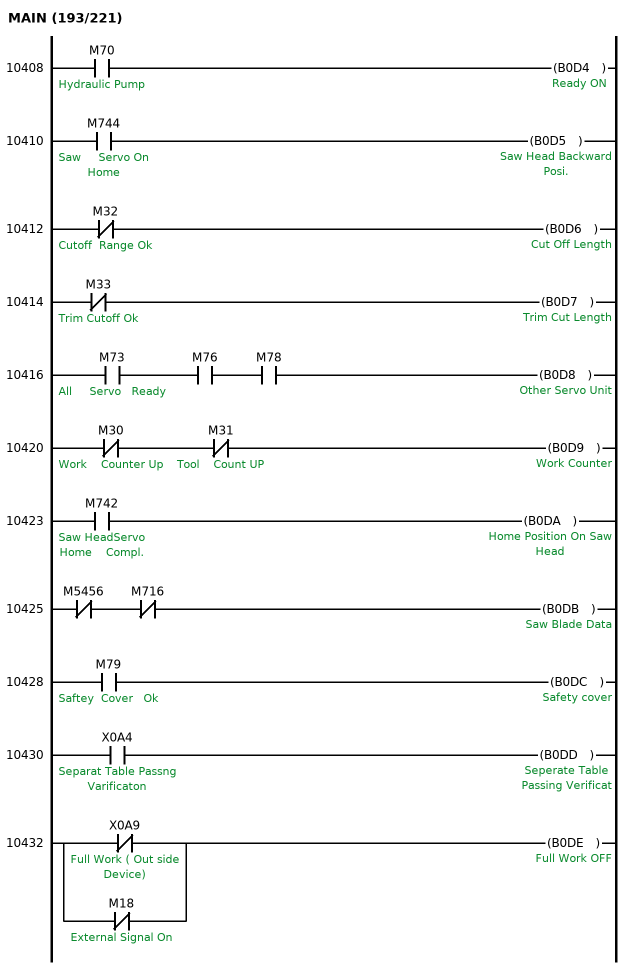
[picture p192: ladder of MAIN, rungs at steps 10408 to 10432]
10408 LD      M70  ; Hydraulic Pump
      OUT     B0D4  ; Ready ON
10410 LD      M744  ; Saw     Servo On Home
      OUT     B0D5  ; Saw Head Backward Posi.
10412 LDI     M32  ; Cutoff  Range Ok
      OUT     B0D6  ; Cut Off Length
10414 LDI     M33  ; Trim Cutoff Ok
      OUT     B0D7  ; Trim Cut Length
10416 LD      M73  ; All     Servo   Ready
      AND     M76
      AND     M78
      OUT     B0D8  ; Other Servo Unit
10420 LDI     M30  ; Work    Counter Up
      ANI     M31  ; Tool    Count UP
      OUT     B0D9  ; Work Counter
10423 LD      M742  ; Saw HeadServo   Home    Compl.
      OUT     B0DA  ; Home Position On Saw Head
10425 LDI     M5456
      ANI     M716
      OUT     B0DB  ; Saw Blade Data
10428 LD      M79  ; Saftey  Cover   Ok
      OUT     B0DC  ; Safety cover
10430 LD      X0A4  ; Separat Table Passng Varificaton
      OUT     B0DD  ; Seperate Table Passing Verificat
10432 LDI     X0A9  ; Full Work ( Out side Device)
      ORI     M18  ; External Signal On
      OUT     B0DE  ; Full Work OFF
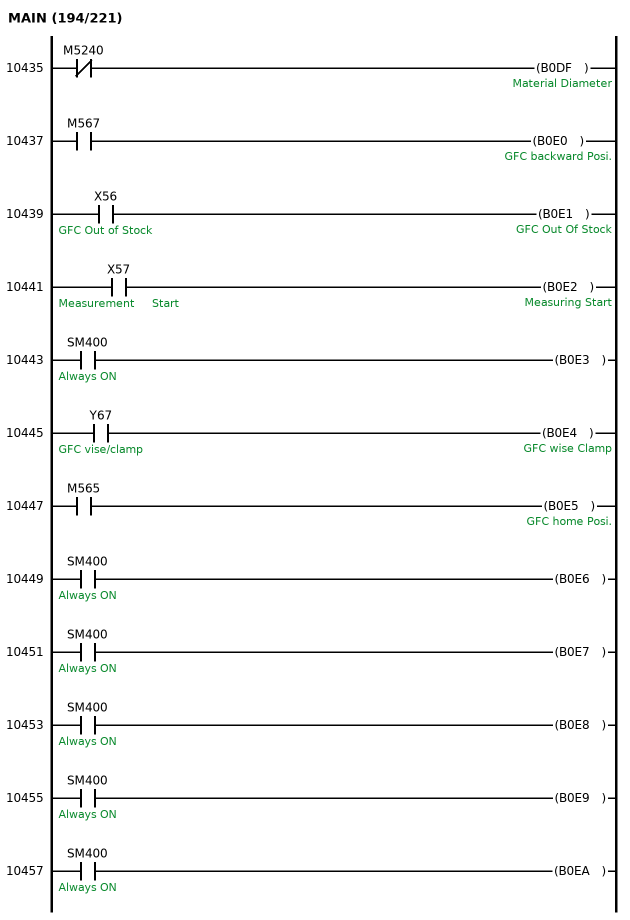
10435 LDI     M5240
      OUT     B0DF  ; Material Diameter
10437 LD      M567
      OUT     B0E0  ; GFC backward Posi.
10439 LD      X56  ; GFC Out of Stock
      OUT     B0E1  ; GFC Out Of Stock
10441 LD      X57  ; Measurement     Start
      OUT     B0E2  ; Measuring Start
10443 LD      SM400  ; Always ON
      OUT     B0E3
10445 LD      Y67  ; GFC vise/clamp
      OUT     B0E4  ; GFC wise Clamp
10447 LD      M565
      OUT     B0E5  ; GFC home Posi.
10449 LD      SM400  ; Always ON
      OUT     B0E6
10451 LD      SM400  ; Always ON
      OUT     B0E7
10453 LD      SM400  ; Always ON
      OUT     B0E8
10455 LD      SM400  ; Always ON
      OUT     B0E9
10457 LD      SM400  ; Always ON
      OUT     B0EA
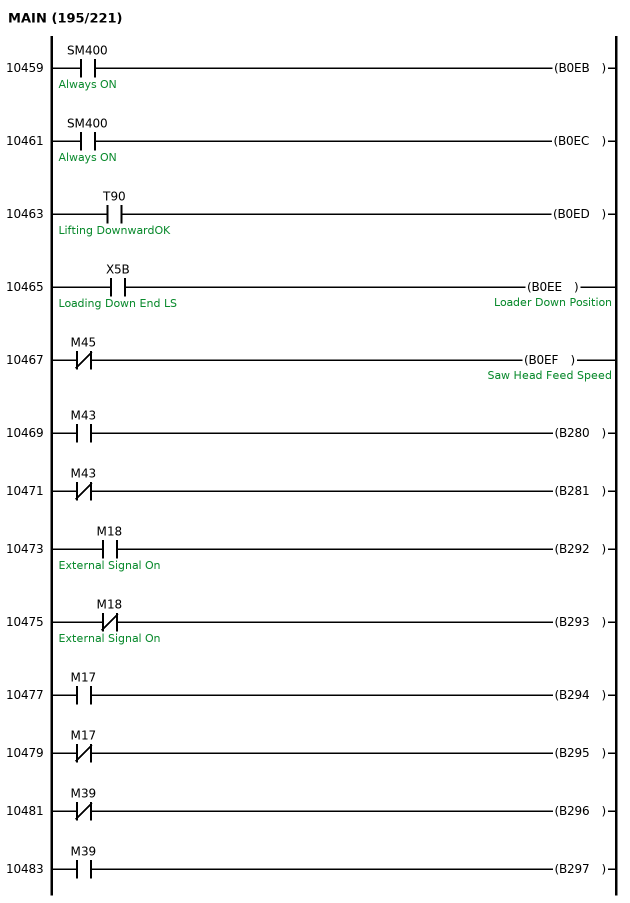
10459 LD      SM400  ; Always ON
      OUT     B0EB
10461 LD      SM400  ; Always ON
      OUT     B0EC
10463 LD      T90  ; Lifting DownwardOK
      OUT     B0ED
10465 LD      X5B  ; Loading Down End LS
      OUT     B0EE  ; Loader Down Position
10467 LDI     M45
      OUT     B0EF  ; Saw Head Feed Speed
10469 LD      M43
      OUT     B280
10471 LDI     M43
      OUT     B281
10473 LD      M18  ; External Signal On
      OUT     B292
10475 LDI     M18  ; External Signal On
      OUT     B293
10477 LD      M17
      OUT     B294
10479 LDI     M17
      OUT     B295
10481 LDI     M39
      OUT     B296
10483 LD      M39
      OUT     B297
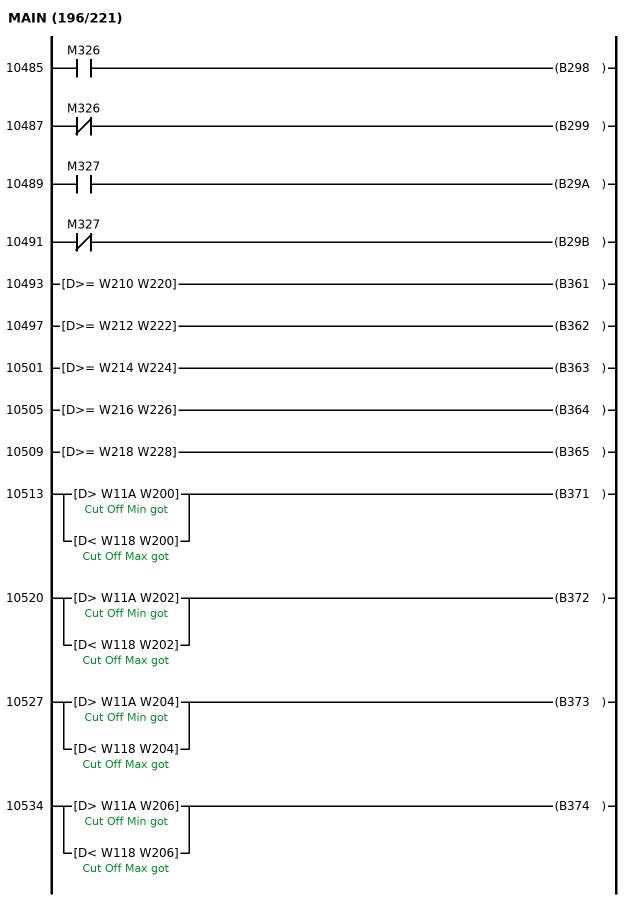
10485 LD      M326
      OUT     B298
10487 LDI     M326
      OUT     B299
10489 LD      M327
      OUT     B29A
10491 LDI     M327
      OUT     B29B
10493 LDD>=   W210 W220
      OUT     B361
10497 LDD>=   W212 W222
      OUT     B362
10501 LDD>=   W214 W224
      OUT     B363
10505 LDD>=   W216 W226
      OUT     B364
10509 LDD>=   W218 W228
      OUT     B365
10513 LDD>    W11A W200  ; Cut Off Min got
      ORD<    W118 W200  ; Cut Off Max got
      OUT     B371
10520 LDD>    W11A W202  ; Cut Off Min got
      ORD<    W118 W202  ; Cut Off Max got
      OUT     B372
10527 LDD>    W11A W204  ; Cut Off Min got
      ORD<    W118 W204  ; Cut Off Max got
      OUT     B373
10534 LDD>    W11A W206  ; Cut Off Min got
      ORD<    W118 W206  ; Cut Off Max got
      OUT     B374
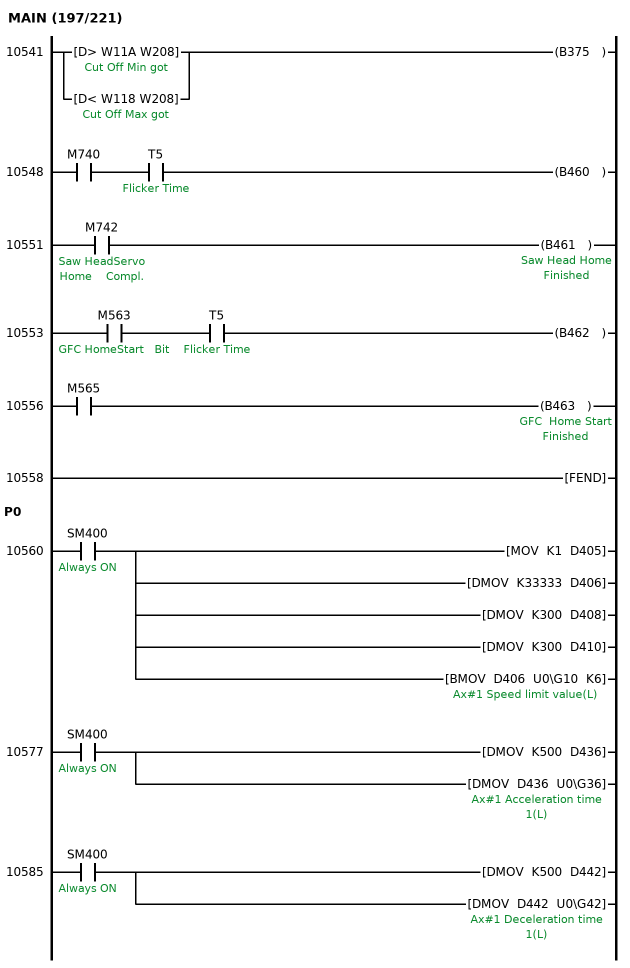
10541 LDD>    W11A W208  ; Cut Off Min got
      ORD<    W118 W208  ; Cut Off Max got
      OUT     B375
10548 LD      M740
      AND     T5  ; Flicker Time
      OUT     B460
10551 LD      M742  ; Saw HeadServo   Home    Compl.
      OUT     B461  ; Saw Head Home Finished
10553 LD      M563  ; GFC HomeStart   Bit
      AND     T5  ; Flicker Time
      OUT     B462
10556 LD      M565
      OUT     B463  ; GFC  Home Start Finished
10558 FEND
      P0
10560 LD      SM400  ; Always ON
      MOV     K1 D405
      DMOV    K33333 D406
      DMOV    K300 D408
      DMOV    K300 D410
      BMOV    D406 U0\G10 K6  ; Ax#1 Speed limit value(L)
10577 LD      SM400  ; Always ON
      DMOV    K500 D436
      DMOV    D436 U0\G36  ; Ax#1 Acceleration time 1(L)
10585 LD      SM400  ; Always ON
      DMOV    K500 D442
      DMOV    D442 U0\G42  ; Ax#1 Deceleration time 1(L)
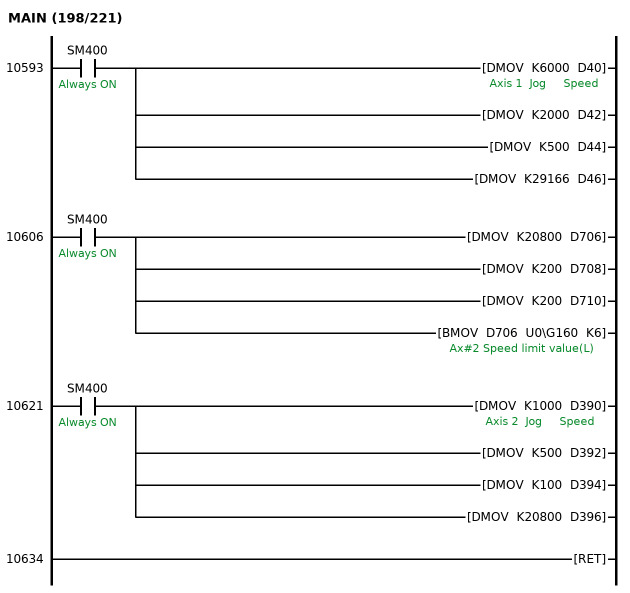
10593 LD      SM400  ; Always ON
      DMOV    K6000 D40
      DMOV    K2000 D42
      DMOV    K500 D44
      DMOV    K29166 D46
10606 LD      SM400  ; Always ON
      DMOV    K20800 D706
      DMOV    K200 D708
      DMOV    K200 D710
      BMOV    D706 U0\G160 K6  ; Ax#2 Speed limit value(L)
10621 LD      SM400  ; Always ON
      DMOV    K1000 D390
      DMOV    K500 D392
      DMOV    K100 D394
      DMOV    K20800 D396
10634 RET
      P1
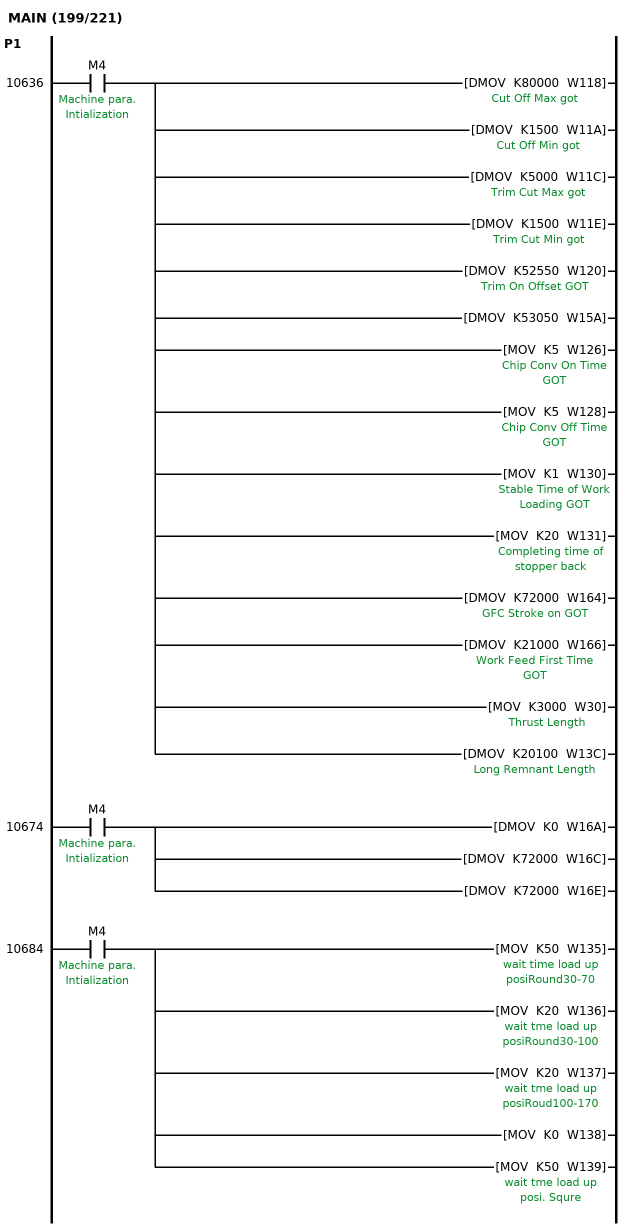
10636 LD      M4  ; Machine para.   Intialization
      DMOV    K80000 W118
      DMOV    K1500 W11A
      DMOV    K5000 W11C
      DMOV    K1500 W11E
      DMOV    K52550 W120
      DMOV    K53050 W15A
      MOV     K5 W126
      MOV     K5 W128
      MOV     K1 W130
      MOV     K20 W131
      DMOV    K72000 W164  ; GFC Stroke on GOT
      DMOV    K21000 W166  ; Work Feed First Time GOT
      MOV     K3000 W30
      DMOV    K20100 W13C
10674 LD      M4  ; Machine para.   Intialization
      DMOV    K0 W16A
      DMOV    K72000 W16C
      DMOV    K72000 W16E
10684 LD      M4  ; Machine para.   Intialization
      MOV     K50 W135
      MOV     K20 W136
      MOV     K20 W137
      MOV     K0 W138
      MOV     K50 W139
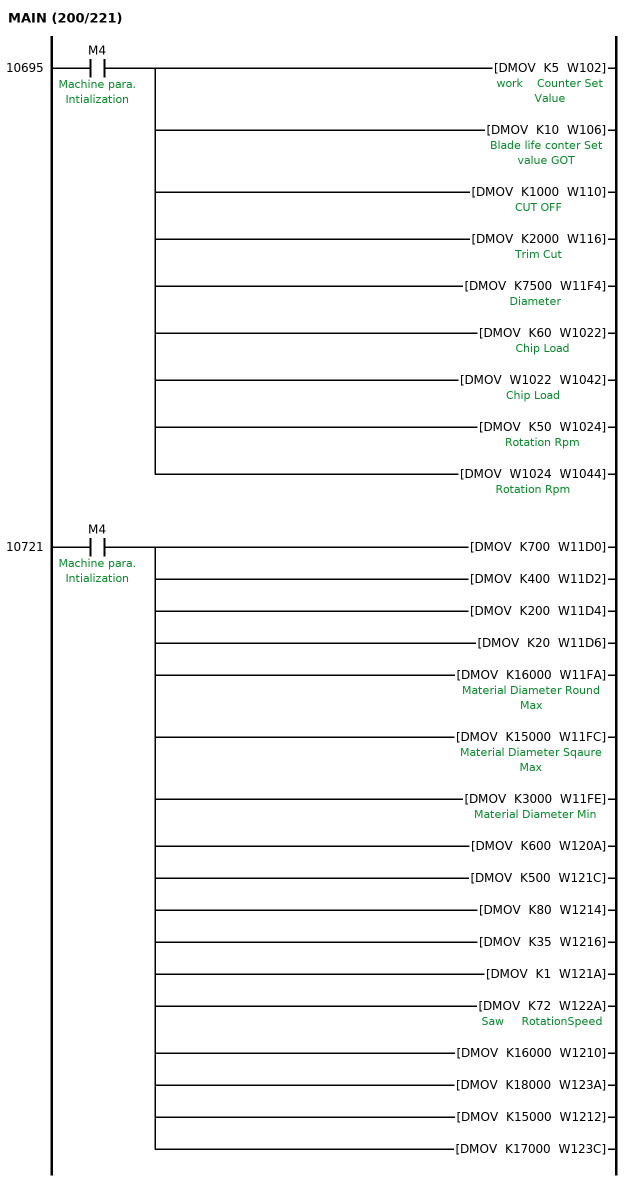
10695 LD      M4  ; Machine para.   Intialization
      DMOV    K5 W102
      DMOV    K10 W106
      DMOV    K1000 W110
      DMOV    K2000 W116
      DMOV    K7500 W11F4
      DMOV    K60 W1022
      DMOV    W1022 W1042
      DMOV    K50 W1024
      DMOV    W1024 W1044
10721 LD      M4  ; Machine para.   Intialization
      DMOV    K700 W11D0
      DMOV    K400 W11D2
      DMOV    K200 W11D4
      DMOV    K20 W11D6
      DMOV    K16000 W11FA
      DMOV    K15000 W11FC
      DMOV    K3000 W11FE
      DMOV    K600 W120A
      DMOV    K500 W121C
      DMOV    K80 W1214
      DMOV    K35 W1216
      DMOV    K1 W121A
      DMOV    K72 W122A
      DMOV    K16000 W1210
      DMOV    K18000 W123A
      DMOV    K15000 W1212
      DMOV    K17000 W123C
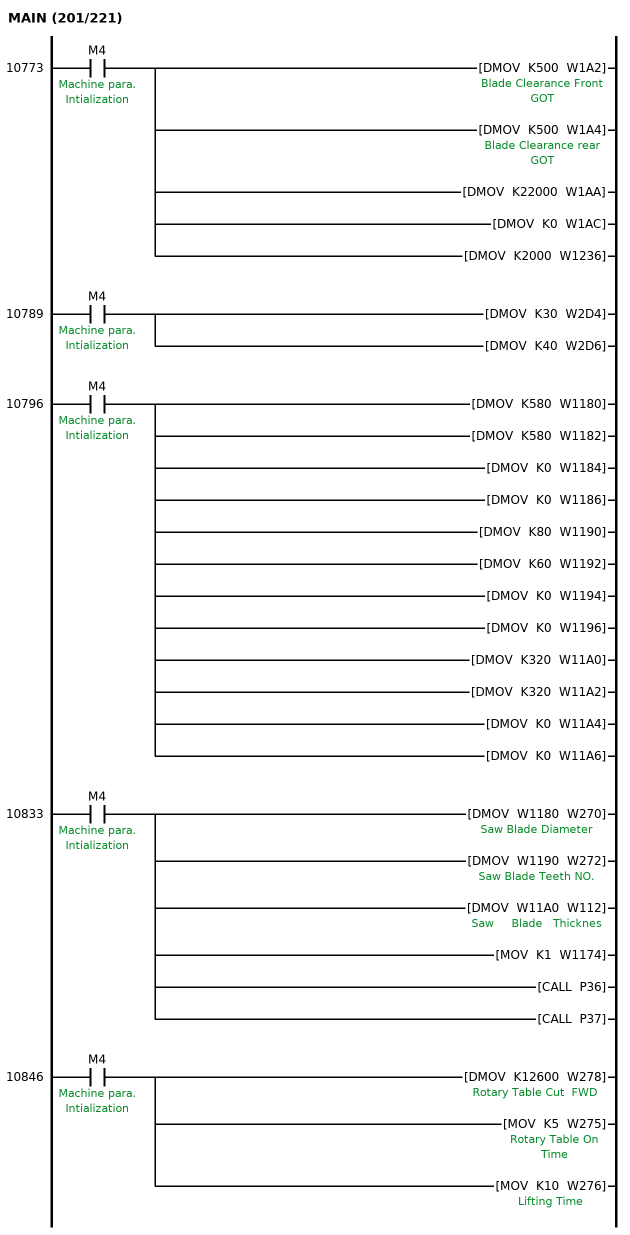
10773 LD      M4  ; Machine para.   Intialization
      DMOV    K500 W1A2
      DMOV    K500 W1A4
      DMOV    K22000 W1AA
      DMOV    K0 W1AC
      DMOV    K2000 W1236
10789 LD      M4  ; Machine para.   Intialization
      DMOV    K30 W2D4
      DMOV    K40 W2D6
10796 LD      M4  ; Machine para.   Intialization
      DMOV    K580 W1180
      DMOV    K580 W1182
      DMOV    K0 W1184
      DMOV    K0 W1186
      DMOV    K80 W1190
      DMOV    K60 W1192
      DMOV    K0 W1194
      DMOV    K0 W1196
      DMOV    K320 W11A0
      DMOV    K320 W11A2
      DMOV    K0 W11A4
      DMOV    K0 W11A6
10833 LD      M4  ; Machine para.   Intialization
      DMOV    W1180 W270
      DMOV    W1190 W272
      DMOV    W11A0 W112
      MOV     K1 W1174
      CALL    P36
      CALL    P37
10846 LD      M4  ; Machine para.   Intialization
      DMOV    K12600 W278
      MOV     K5 W275
      MOV     K10 W276
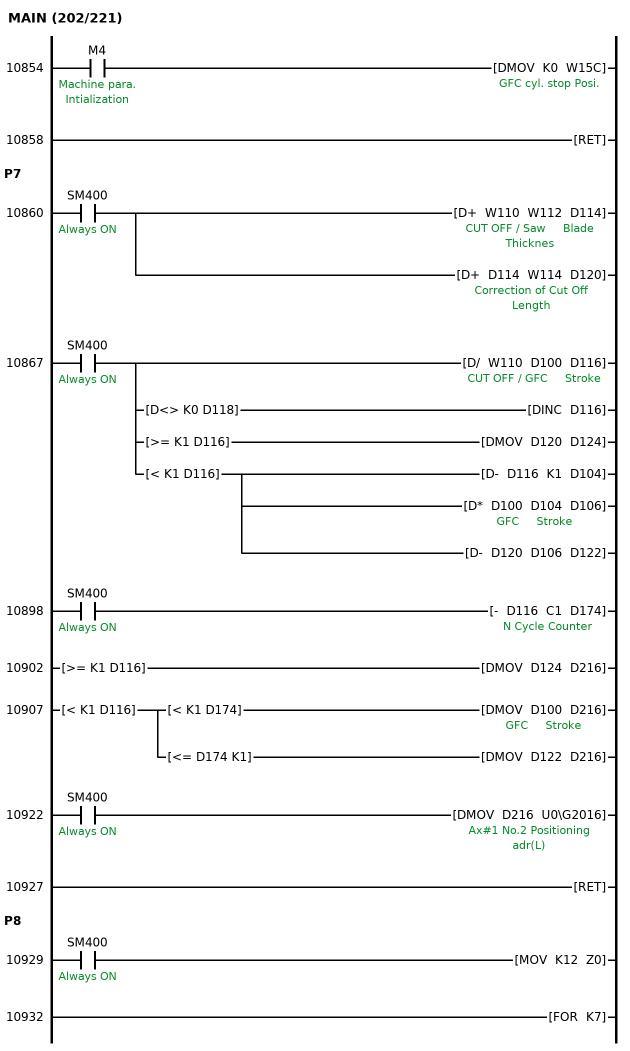
10854 LD      M4  ; Machine para.   Intialization
      DMOV    K0 W15C  ; GFC cyl. stop Posi.
10858 RET
      P7
10860 LD      SM400  ; Always ON
      D+      W110 W112 D114
      D+      D114 W114 D120
10867 LD      SM400  ; Always ON
      D/      W110 D100 D116
      MPS
      ANDD<>  K0 D118
      DINC    D116
      MRD
      AND>=   K1 D116
      DMOV    D120 D124
      MPP
      AND<    K1 D116
      D-      D116 K1 D104
      D*      D100 D104 D106
      D-      D120 D106 D122
10898 LD      SM400  ; Always ON
      -       D116 C1 D174
10902 LD>=    K1 D116
      DMOV    D124 D216
10907 LD<     K1 D116
      MPS
      AND<    K1 D174
      DMOV    D100 D216
      MPP
      AND<=   D174 K1
      DMOV    D122 D216
10922 LD      SM400  ; Always ON
      DMOV    D216 U0\G2016  ; Ax#1 No.2 Positioning adr(L)
10927 RET
      P8
10929 LD      SM400  ; Always ON
      MOV     K12 Z0
10932 FOR     K7
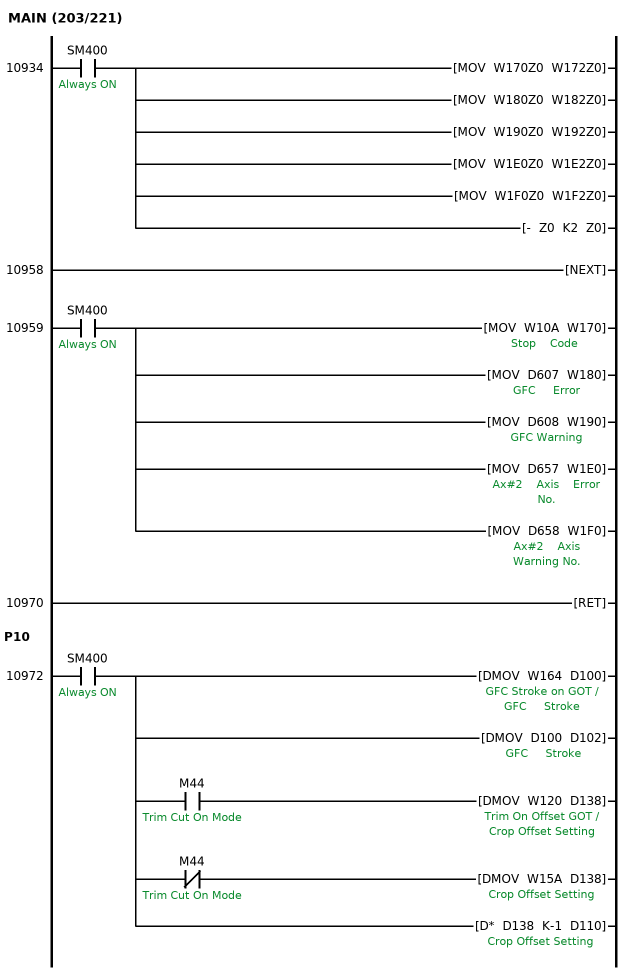
10934 LD      SM400  ; Always ON
      MOV     W170Z0 W172Z0
      MOV     W180Z0 W182Z0
      MOV     W190Z0 W192Z0
      MOV     W1E0Z0 W1E2Z0
      MOV     W1F0Z0 W1F2Z0
      -       Z0 K2 Z0
10958 NEXT
10959 LD      SM400  ; Always ON
      MOV     W10A W170
      MOV     D607 W180
      MOV     D608 W190
      MOV     D657 W1E0
      MOV     D658 W1F0
10970 RET
      P10
10972 LD      SM400  ; Always ON
      DMOV    W164 D100
      DMOV    D100 D102
      MPS
      AND     M44  ; Trim Cut On Mode
      DMOV    W120 D138
      MRD
      ANI     M44  ; Trim Cut On Mode
      DMOV    W15A D138
      MPP
      D*      D138 K-1 D110
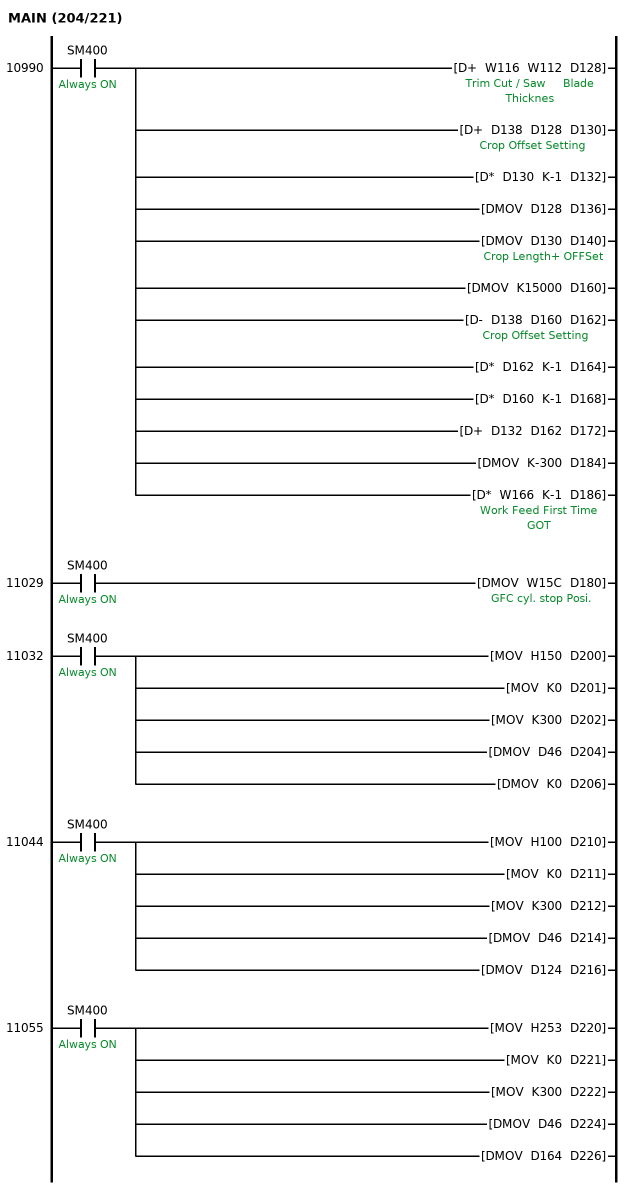
10990 LD      SM400  ; Always ON
      D+      W116 W112 D128
      D+      D138 D128 D130
      D*      D130 K-1 D132
      DMOV    D128 D136
      DMOV    D130 D140
      DMOV    K15000 D160
      D-      D138 D160 D162
      D*      D162 K-1 D164
      D*      D160 K-1 D168
      D+      D132 D162 D172
      DMOV    K-300 D184
      D*      W166 K-1 D186
11029 LD      SM400  ; Always ON
      DMOV    W15C D180
11032 LD      SM400  ; Always ON
      MOV     H150 D200
      MOV     K0 D201
      MOV     K300 D202
      DMOV    D46 D204
      DMOV    K0 D206
11044 LD      SM400  ; Always ON
      MOV     H100 D210
      MOV     K0 D211
      MOV     K300 D212
      DMOV    D46 D214
      DMOV    D124 D216
11055 LD      SM400  ; Always ON
      MOV     H253 D220
      MOV     K0 D221
      MOV     K300 D222
      DMOV    D46 D224
      DMOV    D164 D226
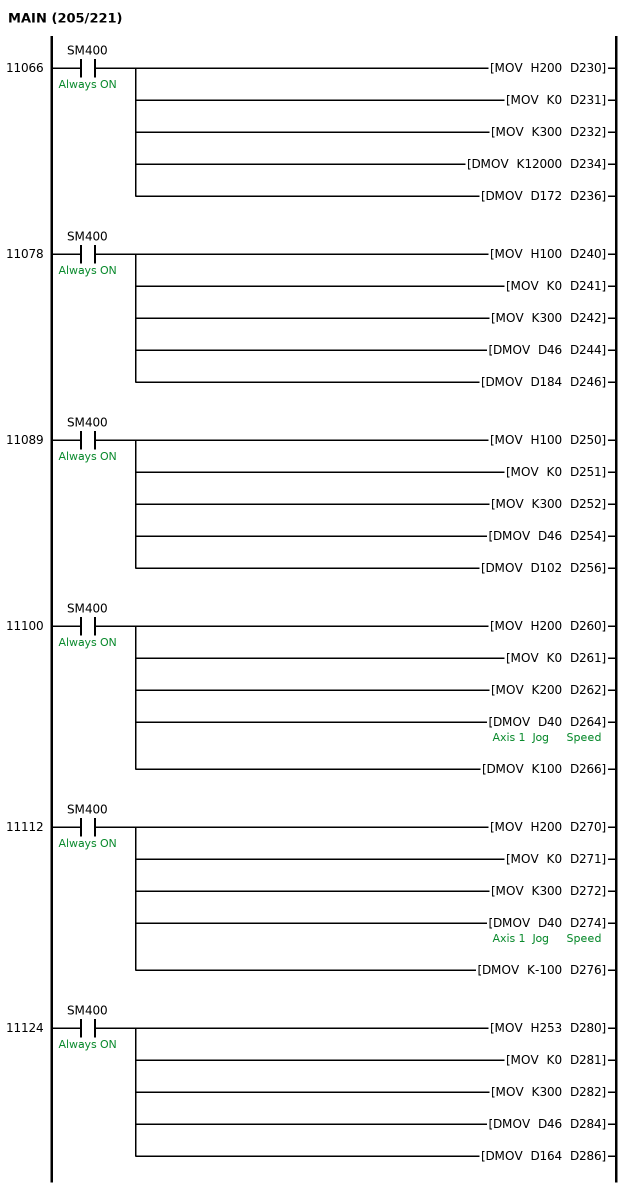
11066 LD      SM400  ; Always ON
      MOV     H200 D230
      MOV     K0 D231
      MOV     K300 D232
      DMOV    K12000 D234
      DMOV    D172 D236
11078 LD      SM400  ; Always ON
      MOV     H100 D240
      MOV     K0 D241
      MOV     K300 D242
      DMOV    D46 D244
      DMOV    D184 D246
11089 LD      SM400  ; Always ON
      MOV     H100 D250
      MOV     K0 D251
      MOV     K300 D252
      DMOV    D46 D254
      DMOV    D102 D256
11100 LD      SM400  ; Always ON
      MOV     H200 D260
      MOV     K0 D261
      MOV     K200 D262
      DMOV    D40 D264
      DMOV    K100 D266
11112 LD      SM400  ; Always ON
      MOV     H200 D270
      MOV     K0 D271
      MOV     K300 D272
      DMOV    D40 D274
      DMOV    K-100 D276
11124 LD      SM400  ; Always ON
      MOV     H253 D280
      MOV     K0 D281
      MOV     K300 D282
      DMOV    D46 D284
      DMOV    D164 D286
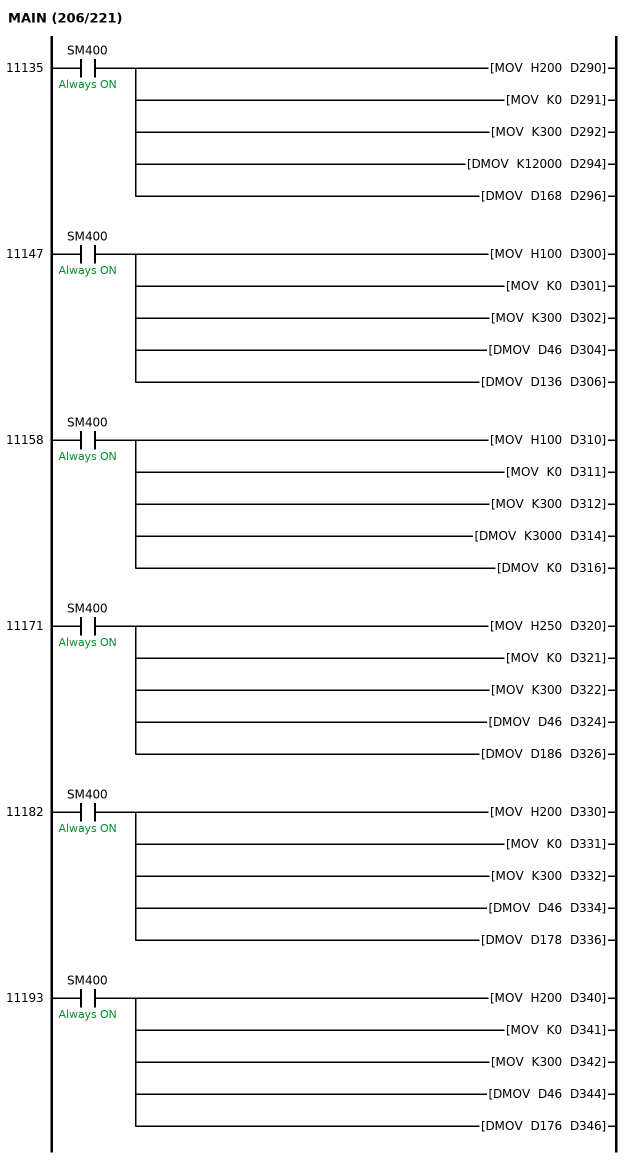
11135 LD      SM400  ; Always ON
      MOV     H200 D290
      MOV     K0 D291
      MOV     K300 D292
      DMOV    K12000 D294
      DMOV    D168 D296
11147 LD      SM400  ; Always ON
      MOV     H100 D300
      MOV     K0 D301
      MOV     K300 D302
      DMOV    D46 D304
      DMOV    D136 D306
11158 LD      SM400  ; Always ON
      MOV     H100 D310
      MOV     K0 D311
      MOV     K300 D312
      DMOV    K3000 D314
      DMOV    K0 D316
11171 LD      SM400  ; Always ON
      MOV     H250 D320
      MOV     K0 D321
      MOV     K300 D322
      DMOV    D46 D324
      DMOV    D186 D326
11182 LD      SM400  ; Always ON
      MOV     H200 D330
      MOV     K0 D331
      MOV     K300 D332
      DMOV    D46 D334
      DMOV    D178 D336
11193 LD      SM400  ; Always ON
      MOV     H200 D340
      MOV     K0 D341
      MOV     K300 D342
      DMOV    D46 D344
      DMOV    D176 D346
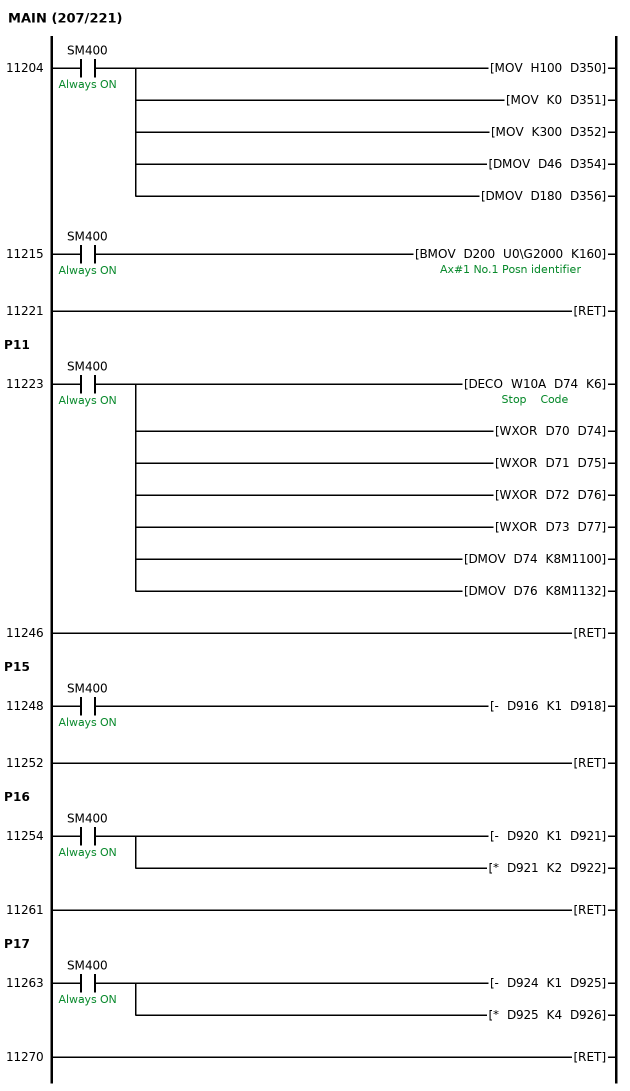
11204 LD      SM400  ; Always ON
      MOV     H100 D350
      MOV     K0 D351
      MOV     K300 D352
      DMOV    D46 D354
      DMOV    D180 D356
11215 LD      SM400  ; Always ON
      BMOV    D200 U0\G2000 K160  ; Ax#1 No.1 Posn identifier
11221 RET
      P11
11223 LD      SM400  ; Always ON
      DECO    W10A D74 K6
      WXOR    D70 D74
      WXOR    D71 D75
      WXOR    D72 D76
      WXOR    D73 D77
      DMOV    D74 K8M1100
      DMOV    D76 K8M1132
11246 RET
      P15
11248 LD      SM400  ; Always ON
      -       D916 K1 D918
11252 RET
      P16
11254 LD      SM400  ; Always ON
      -       D920 K1 D921
      *       D921 K2 D922
11261 RET
      P17
11263 LD      SM400  ; Always ON
      -       D924 K1 D925
      *       D925 K4 D926
11270 RET
      P21
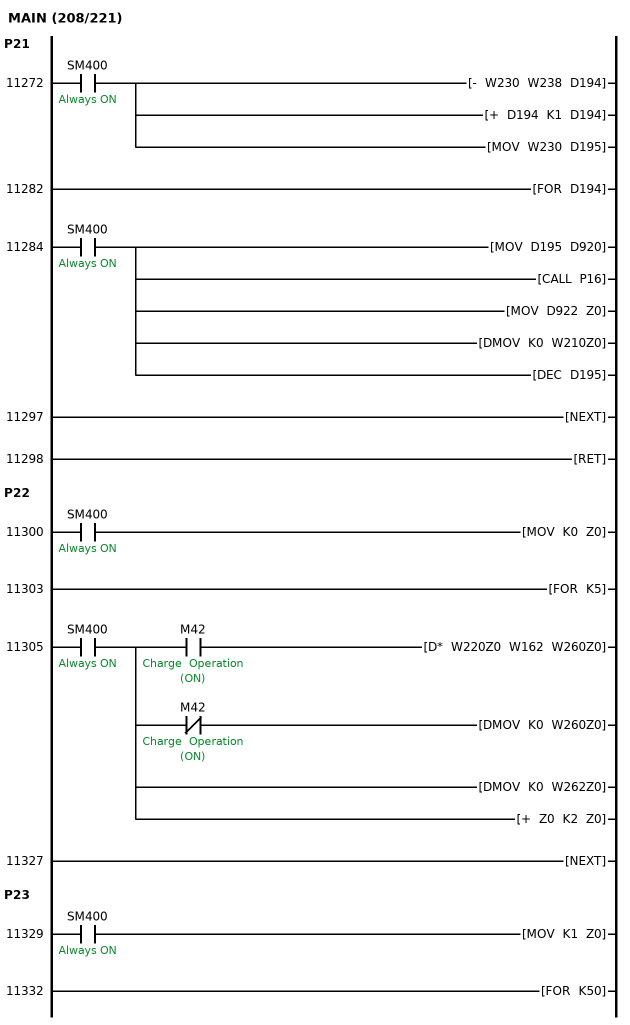
11272 LD      SM400  ; Always ON
      -       W230 W238 D194
      +       D194 K1 D194
      MOV     W230 D195
11282 FOR     D194
11284 LD      SM400  ; Always ON
      MOV     D195 D920
      CALL    P16
      MOV     D922 Z0
      DMOV    K0 W210Z0
      DEC     D195
11297 NEXT
11298 RET
      P22
11300 LD      SM400  ; Always ON
      MOV     K0 Z0
11303 FOR     K5
11305 LD      SM400  ; Always ON
      MPS
      AND     M42  ; Charge  Operation (ON)
      D*      W220Z0 W162 W260Z0
      MRD
      ANI     M42  ; Charge  Operation (ON)
      DMOV    K0 W260Z0
      MPP
      DMOV    K0 W262Z0
      +       Z0 K2 Z0
11327 NEXT
      P23
11329 LD      SM400  ; Always ON
      MOV     K1 Z0
11332 FOR     K50
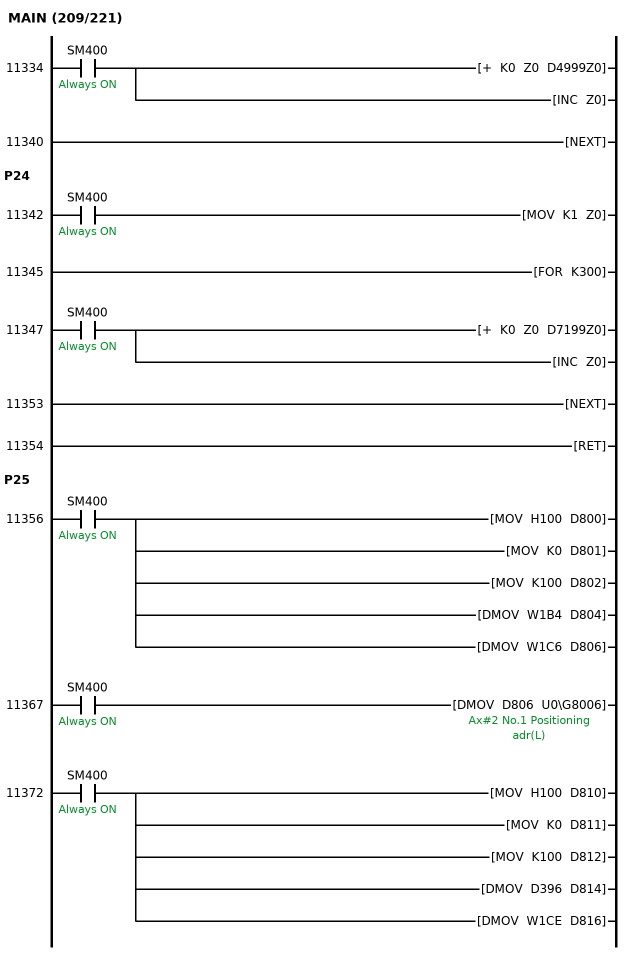
11334 LD      SM400  ; Always ON
      +       K0 Z0 D4999Z0
      INC     Z0
11340 NEXT
      P24
11342 LD      SM400  ; Always ON
      MOV     K1 Z0
11345 FOR     K300
11347 LD      SM400  ; Always ON
      +       K0 Z0 D7199Z0
      INC     Z0
11353 NEXT
11354 RET
      P25
11356 LD      SM400  ; Always ON
      MOV     H100 D800
      MOV     K0 D801
      MOV     K100 D802
      DMOV    W1B4 D804
      DMOV    W1C6 D806
11367 LD      SM400  ; Always ON
      DMOV    D806 U0\G8006  ; Ax#2 No.1 Positioning adr(L)
11372 LD      SM400  ; Always ON
      MOV     H100 D810
      MOV     K0 D811
      MOV     K100 D812
      DMOV    D396 D814
      DMOV    W1CE D816
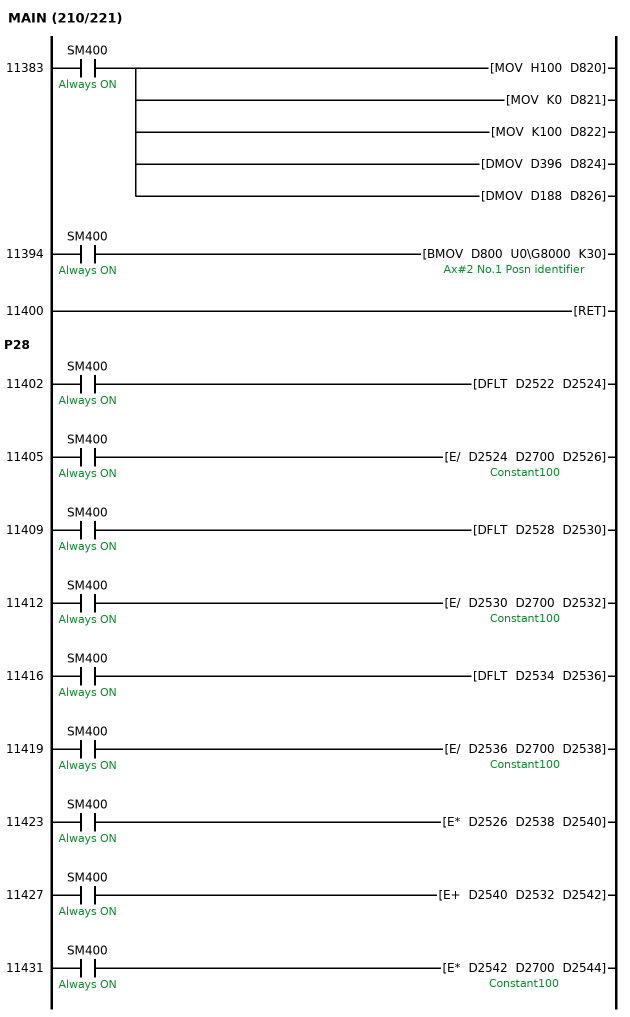
11383 LD      SM400  ; Always ON
      MOV     H100 D820
      MOV     K0 D821
      MOV     K100 D822
      DMOV    D396 D824
      DMOV    D188 D826
11394 LD      SM400  ; Always ON
      BMOV    D800 U0\G8000 K30  ; Ax#2 No.1 Posn identifier
11400 RET
      P28
11402 LD      SM400  ; Always ON
      DFLT    D2522 D2524
11405 LD      SM400  ; Always ON
      E/      D2524 D2700 D2526  ; Constant100
11409 LD      SM400  ; Always ON
      DFLT    D2528 D2530
11412 LD      SM400  ; Always ON
      E/      D2530 D2700 D2532
11416 LD      SM400  ; Always ON
      DFLT    D2534 D2536
11419 LD      SM400  ; Always ON
      E/      D2536 D2700 D2538
11423 LD      SM400  ; Always ON
      E*      D2526 D2538 D2540
11427 LD      SM400  ; Always ON
      E+      D2540 D2532 D2542
11431 LD      SM400  ; Always ON
      E*      D2542 D2700 D2544
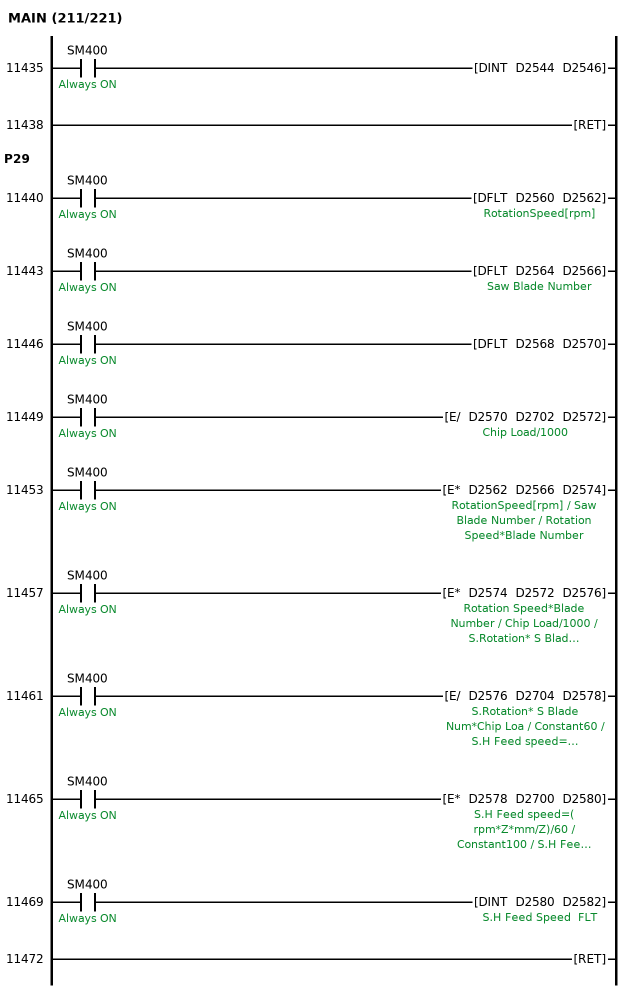
11435 LD      SM400  ; Always ON
      DINT    D2544 D2546
11438 RET
      P29
11440 LD      SM400  ; Always ON
      DFLT    D2560 D2562  ; RotationSpeed[rpm]
11443 LD      SM400  ; Always ON
      DFLT    D2564 D2566  ; Saw Blade Number
11446 LD      SM400  ; Always ON
      DFLT    D2568 D2570
11449 LD      SM400  ; Always ON
      E/      D2570 D2702 D2572  ; Chip Load/1000
11453 LD      SM400  ; Always ON
      E*      D2562 D2566 D2574  ; Rotation Speed*Blade Number
11457 LD      SM400  ; Always ON
      E*      D2574 D2572 D2576  ; S.Rotation* S Blade Num*Chip Loa
11461 LD      SM400  ; Always ON
      E/      D2576 D2704 D2578  ; Constant60 / S.H Feed speed=(rpm*Z*mm/Z)/60
11465 LD      SM400  ; Always ON
      E*      D2578 D2700 D2580  ; S.H Feed Speed  FLT
11469 LD      SM400  ; Always ON
      DINT    D2580 D2582
11472 RET
      P31
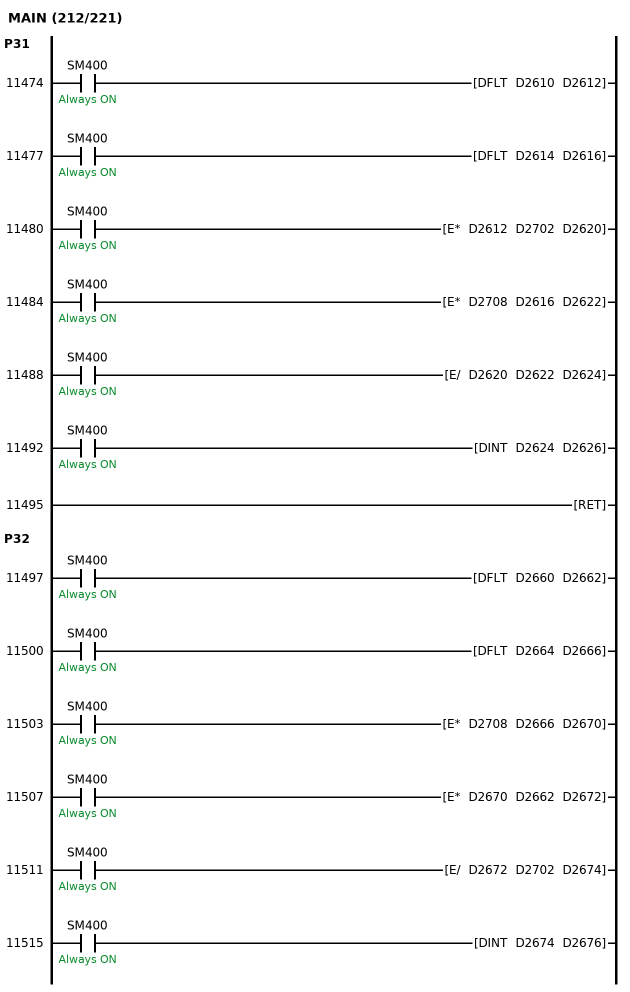
11474 LD      SM400  ; Always ON
      DFLT    D2610 D2612
11477 LD      SM400  ; Always ON
      DFLT    D2614 D2616
11480 LD      SM400  ; Always ON
      E*      D2612 D2702 D2620
11484 LD      SM400  ; Always ON
      E*      D2708 D2616 D2622
11488 LD      SM400  ; Always ON
      E/      D2620 D2622 D2624
11492 LD      SM400  ; Always ON
      DINT    D2624 D2626
11495 RET
      P32
11497 LD      SM400  ; Always ON
      DFLT    D2660 D2662
11500 LD      SM400  ; Always ON
      DFLT    D2664 D2666
11503 LD      SM400  ; Always ON
      E*      D2708 D2666 D2670
11507 LD      SM400  ; Always ON
      E*      D2670 D2662 D2672
11511 LD      SM400  ; Always ON
      E/      D2672 D2702 D2674
11515 LD      SM400  ; Always ON
      DINT    D2674 D2676
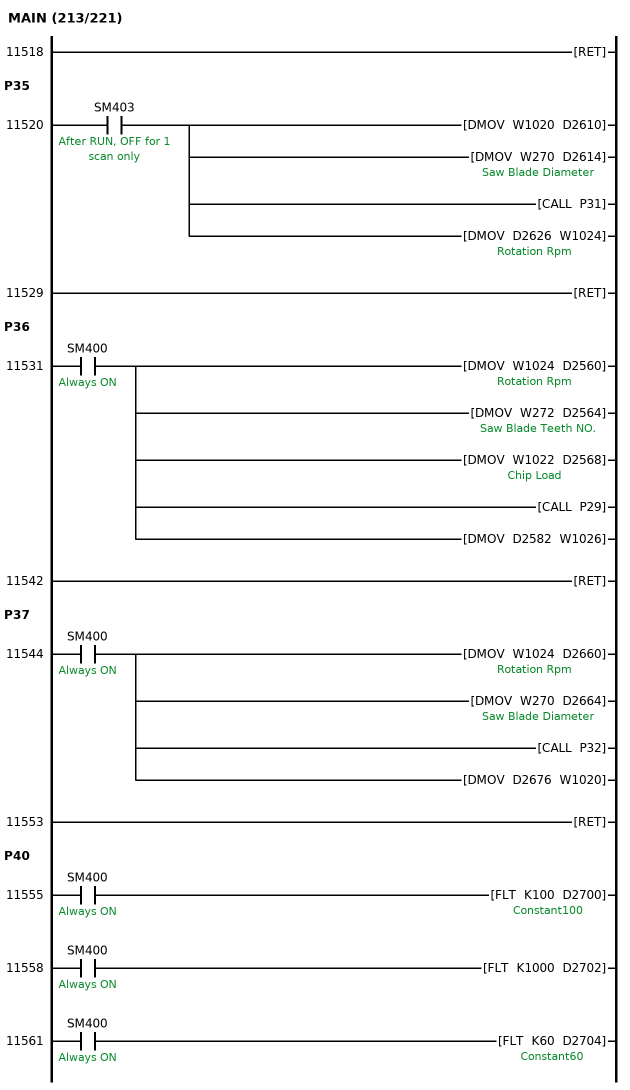
11518 RET
      P35
11520 LD      SM403  ; After RUN, OFF for 1 scan only
      DMOV    W1020 D2610
      DMOV    W270 D2614
      CALL    P31
      DMOV    D2626 W1024
11529 RET
      P36
11531 LD      SM400  ; Always ON
      DMOV    W1024 D2560
      DMOV    W272 D2564
      DMOV    W1022 D2568
      CALL    P29
      DMOV    D2582 W1026
11542 RET
      P37
11544 LD      SM400  ; Always ON
      DMOV    W1024 D2660
      DMOV    W270 D2664
      CALL    P32
      DMOV    D2676 W1020
11553 RET
      P40
11555 LD      SM400  ; Always ON
      FLT     K100 D2700
11558 LD      SM400  ; Always ON
      FLT     K1000 D2702
11561 LD      SM400  ; Always ON
      FLT     K60 D2704
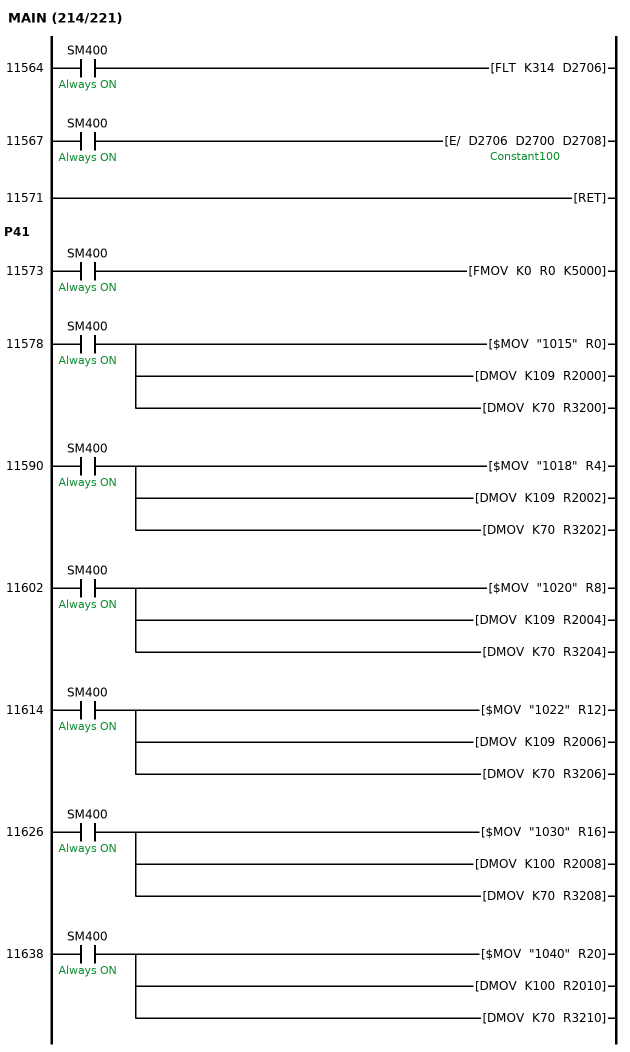
11564 LD      SM400  ; Always ON
      FLT     K314 D2706
11567 LD      SM400  ; Always ON
      E/      D2706 D2700 D2708
11571 RET
      P41
11573 LD      SM400  ; Always ON
      FMOV    K0 R0 K5000
11578 LD      SM400  ; Always ON
      $MOV    "1015" R0
      DMOV    K109 R2000
      DMOV    K70 R3200
11590 LD      SM400  ; Always ON
      $MOV    "1018" R4
      DMOV    K109 R2002
      DMOV    K70 R3202
11602 LD      SM400  ; Always ON
      $MOV    "1020" R8
      DMOV    K109 R2004
      DMOV    K70 R3204
11614 LD      SM400  ; Always ON
      $MOV    "1022" R12
      DMOV    K109 R2006
      DMOV    K70 R3206
11626 LD      SM400  ; Always ON
      $MOV    "1030" R16
      DMOV    K100 R2008
      DMOV    K70 R3208
11638 LD      SM400  ; Always ON
      $MOV    "1040" R20
      DMOV    K100 R2010
      DMOV    K70 R3210
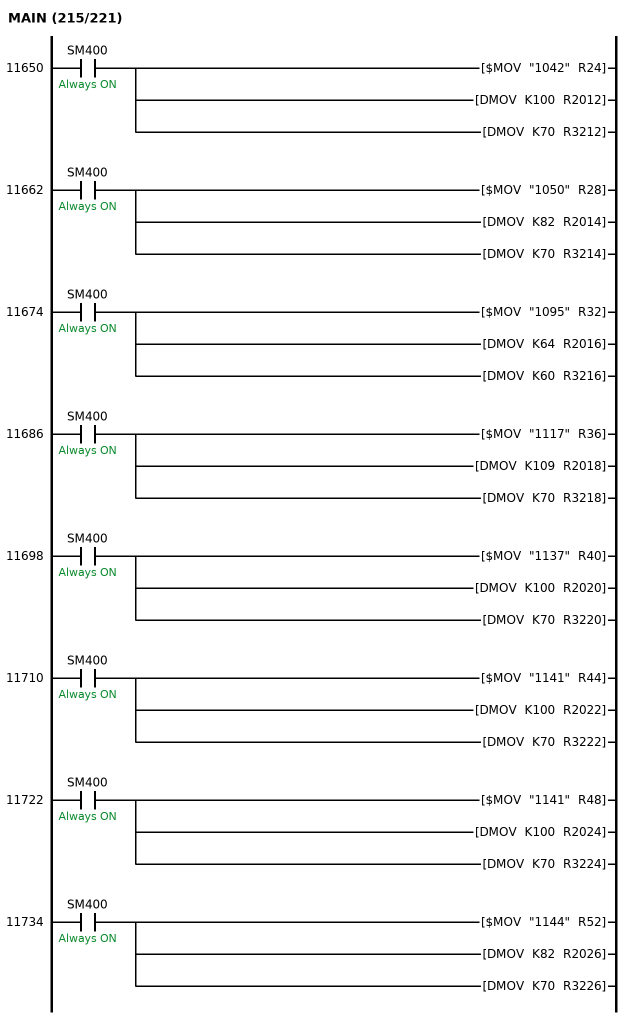
11650 LD      SM400  ; Always ON
      $MOV    "1042" R24
      DMOV    K100 R2012
      DMOV    K70 R3212
11662 LD      SM400  ; Always ON
      $MOV    "1050" R28
      DMOV    K82 R2014
      DMOV    K70 R3214
11674 LD      SM400  ; Always ON
      $MOV    "1095" R32
      DMOV    K64 R2016
      DMOV    K60 R3216
11686 LD      SM400  ; Always ON
      $MOV    "1117" R36
      DMOV    K109 R2018
      DMOV    K70 R3218
11698 LD      SM400  ; Always ON
      $MOV    "1137" R40
      DMOV    K100 R2020
      DMOV    K70 R3220
11710 LD      SM400  ; Always ON
      $MOV    "1141" R44
      DMOV    K100 R2022
      DMOV    K70 R3222
11722 LD      SM400  ; Always ON
      $MOV    "1141" R48
      DMOV    K100 R2024
      DMOV    K70 R3224
11734 LD      SM400  ; Always ON
      $MOV    "1144" R52
      DMOV    K82 R2026
      DMOV    K70 R3226
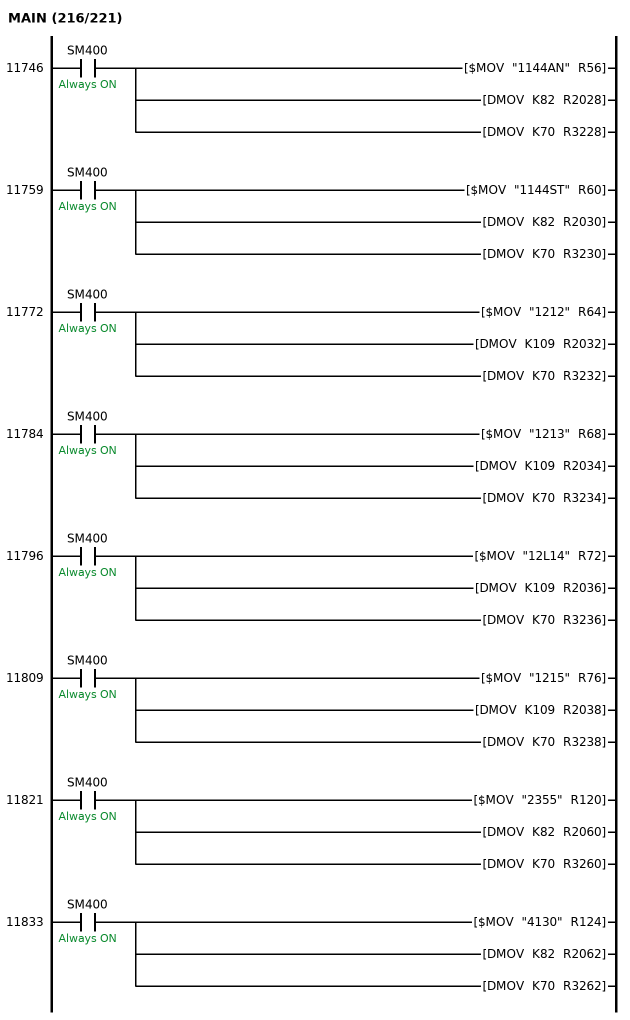
11746 LD      SM400  ; Always ON
      $MOV    "1144AN" R56
      DMOV    K82 R2028
      DMOV    K70 R3228
11759 LD      SM400  ; Always ON
      $MOV    "1144ST" R60
      DMOV    K82 R2030
      DMOV    K70 R3230
11772 LD      SM400  ; Always ON
      $MOV    "1212" R64
      DMOV    K109 R2032
      DMOV    K70 R3232
11784 LD      SM400  ; Always ON
      $MOV    "1213" R68
      DMOV    K109 R2034
      DMOV    K70 R3234
11796 LD      SM400  ; Always ON
      $MOV    "12L14" R72
      DMOV    K109 R2036
      DMOV    K70 R3236
11809 LD      SM400  ; Always ON
      $MOV    "1215" R76
      DMOV    K109 R2038
      DMOV    K70 R3238
11821 LD      SM400  ; Always ON
      $MOV    "2355" R120
      DMOV    K82 R2060
      DMOV    K70 R3260
11833 LD      SM400  ; Always ON
      $MOV    "4130" R124
      DMOV    K82 R2062
      DMOV    K70 R3262
